{attribute addProperty BoxType "AT2026-0250-0022"}
{attribute addProperty Id "A_0079_AT2002_5249_0018_AT2002_5249AT2002_3DCFC8D064080"}
{attribute addProperty CRC "3635088611"}
{attribute addProperty SizeInBites "640"}
{attribute addProperty SizeInBytes "80"}
TYPE A_0067_AT2026_0250_0022_AT2026_0250_D8AB0CE3 EXTENDS AT2026_9506A482 :
STRUCT
	{attribute addProperty Name "A_0079_AT2002_5249_0018_AT2002_5249"}
	A_0079_AT2002_5249_0018_AT2002_5249 : AT2002_3DCFC8D0;
END_STRUCT
END_TYPE

(* stored: Version 1.2.0.0, ProductVersion 3.1.4024.9
   DUT A_0067_AT2026_0250_0022_AT2026_0250_D8AB0CE3: Id {b5ae6a83-d3bf-4b9b-bdb2-a3eb593cd344} *)
